FUNCTION_BLOCK FB_BlueDiverter EXTENDS FB_BaseDiverter
VAR_INPUT
END_VAR
VAR_OUTPUT
END_VAR
VAR
END_VAR

METHOD PUBLIC Sort
VAR_INPUT
    color : E_Color;
END_VAR
IF color = E_Color.BLUE THEN
    Start();
END_IF
END_METHOD

END_FUNCTION_BLOCK

(* stored: Version 1.1.0.1
   POU FB_BlueDiverter: Id {17d30996-a73b-4b18-9eb8-be7fe6182d8a}, SpecialFunc None
   Method Sort: Id {e325922e-9899-40ef-84bb-78d6b94a08f2} *)
